INTERFACE I_TermFuse

PROPERTY IsActive : BOOL
GET
END_GET
END_PROPERTY

END_INTERFACE

(* stored: Version 1.1.0.1, ProductVersion 3.1.4024.12
   Itf I_TermFuse: Id {0573ceee-50ba-429c-b51a-a4dd1cf710ff}
   Property IsActive: Id {c2383986-bf17-437f-8b08-8d0280441366}
   Get Get: Id {75b0de78-b082-4195-b620-8ef0e3350276} *)
